// Mitsubishi GX Works2 project: 0710-DA전압2   PLC: Q02/Q02H

PROGRAM MAIN
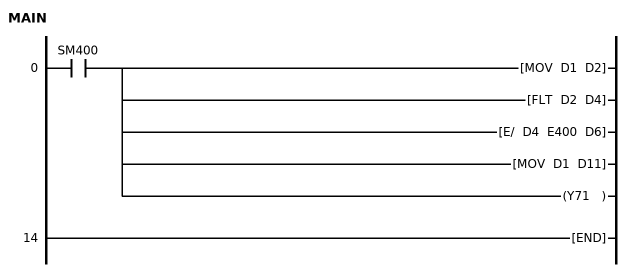
0     LD      SM400
      MOV     D1 D2
      FLT     D2 D4
      E/      D4 E400 D6
      MOV     D1 D11
      OUT     Y71
14    END
END_PROGRAM
